FUNCTION_BLOCK ConveyorCTLMulticast (* Basic Function Block Type *)
  (* Standard: 61499-2 *)
  (* Version 0.2, 2003-12-04, JHC, Rockwell Automation, Renamed for better indexing. *)
  (* Version 0.1, 2002-11-05, JHC, Rockwell Automation, Corrected missing ST element in Algorithm REQ. *)
  (* Version 0.0, 2000-05-30, JHC, Rockwell Automation *)
  (* Compiler header: package fb.rt.cs725; *)
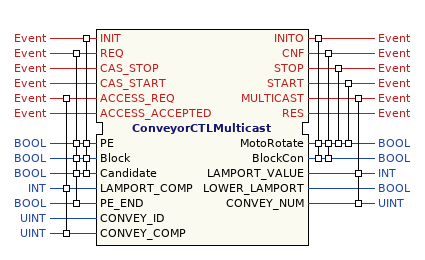
  EVENT_INPUT
    INIT WITH PE, Block, Candidate; (* Initialization Request *)
    REQ WITH PE, Block, Candidate, PE_END; (* Normal Execution Request *)
    CAS_STOP;
    CAS_START;
    ACCESS_REQ WITH LAMPORT_COMP, CONVEY_COMP;
    ACCESS_ACCEPTED;
  END_EVENT
  EVENT_OUTPUT
    INITO WITH MotoRotate, BlockCon; (* Initialization Confirm *)
    CNF WITH MotoRotate, BlockCon; (* Execution Confirmation *)
    STOP WITH MotoRotate;
    START WITH MotoRotate;
    MULTICAST WITH LAMPORT_VALUE, CONVEY_NUM;
    RES;
  END_EVENT
  VAR_INPUT
    PE : BOOL; (* Input event qualifier *)
    Block : BOOL;
    Candidate : BOOL;
    LAMPORT_COMP : INT;
    PE_END : BOOL;
    CONVEY_ID : UINT;
    CONVEY_COMP : UINT;
  END_VAR
  VAR_OUTPUT
    MotoRotate : BOOL; (* Output event qualifier *)
    BlockCon : BOOL;
    LAMPORT_VALUE : INT;
    LOWER_LAMPORT : BOOL;
    CONVEY_NUM : UINT;
  END_VAR
  VAR
    lastPE : BOOL := 1;
    lastBlock : BOOL := 0;
    LAMPORT_CLOCK : INT := 0;
  END_VAR
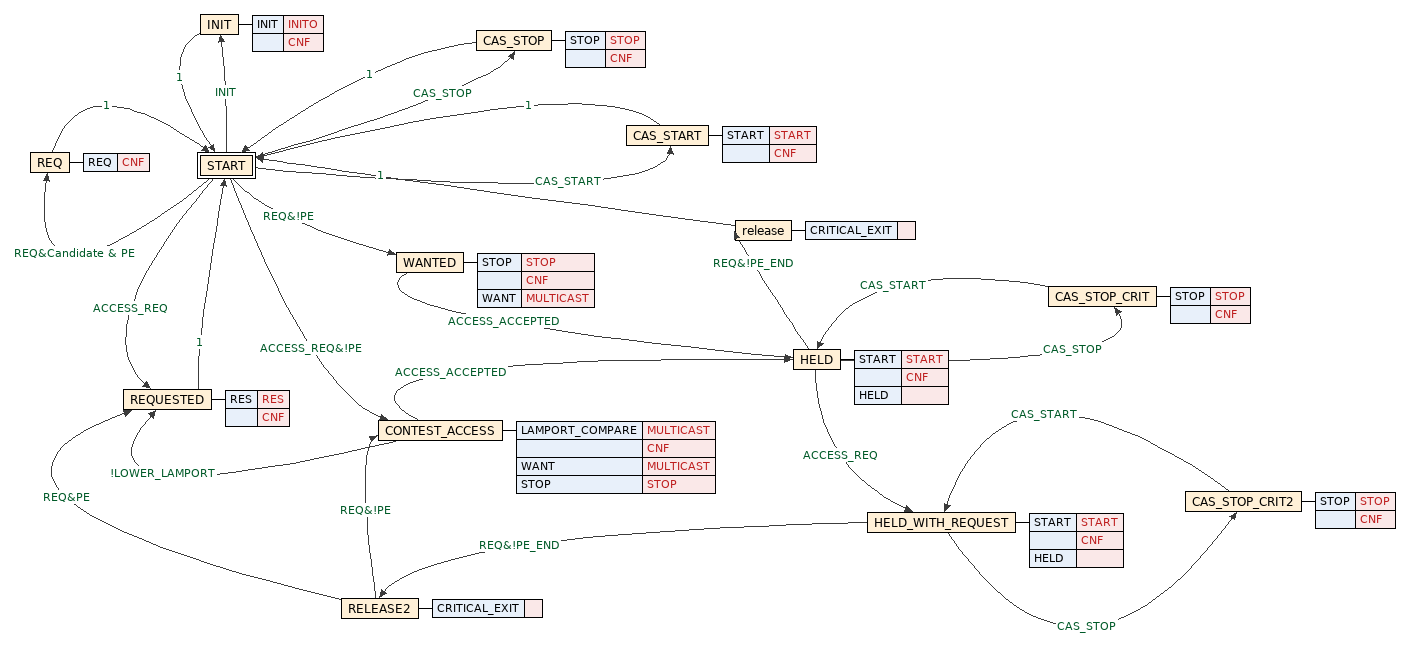
  EC_STATES
    START; (* Initial State *)
    INIT : INIT -> INITO, -> CNF; (* Initialization *)
    REQ : REQ -> CNF; (* Normal execution *)
    CAS_START : START -> START, -> CNF;
    CAS_STOP : STOP -> STOP, -> CNF;
    WANTED : STOP -> STOP, -> CNF, WANT -> MULTICAST;
    HELD : START -> START, -> CNF, HELD;
    REQUESTED : RES -> RES, -> CNF;
    CAS_STOP_CRIT : STOP -> STOP, -> CNF;
    CONTEST_ACCESS : LAMPORT_COMPARE -> MULTICAST, -> CNF, WANT -> MULTICAST, STOP -> STOP;
    release : CRITICAL_EXIT;
    HELD_WITH_REQUEST : START -> START, -> CNF, HELD;
    RELEASE2 : CRITICAL_EXIT;
    CAS_STOP_CRIT2 : STOP -> STOP, -> CNF;
  END_STATES
  EC_TRANSITIONS
    START TO INIT := INIT;
    INIT TO START := 1;
    START TO REQ := REQ&Candidate & PE;
    REQ TO START := 1;
    START TO CAS_START := CAS_START;
    CAS_START TO START := 1;
    START TO CAS_STOP := CAS_STOP;
    CAS_STOP TO START := 1;
    WANTED TO HELD := ACCESS_ACCEPTED;
    START TO WANTED := REQ&!PE;
    START TO REQUESTED := ACCESS_REQ;
    REQUESTED TO START := 1;
    CAS_STOP_CRIT TO HELD := CAS_START;
    START TO CONTEST_ACCESS := ACCESS_REQ&!PE;
    CONTEST_ACCESS TO REQUESTED := !LOWER_LAMPORT;
    CONTEST_ACCESS TO HELD := ACCESS_ACCEPTED;
    release TO START := 1;
    HELD TO release := REQ&!PE_END;
    HELD TO CAS_STOP_CRIT := CAS_STOP;
    HELD TO HELD_WITH_REQUEST := ACCESS_REQ;
    HELD_WITH_REQUEST TO CAS_STOP_CRIT2 := CAS_STOP;
    CAS_STOP_CRIT2 TO HELD_WITH_REQUEST := CAS_START;
    HELD_WITH_REQUEST TO RELEASE2 := REQ&!PE_END;
    RELEASE2 TO CONTEST_ACCESS := REQ&!PE;
    RELEASE2 TO REQUESTED := REQ&PE;
  END_TRANSITIONS
  ALGORITHM INIT IN ST: (* Initialization algorithm *)
MotoRotate := TRUE;
Block := FALSE;

System.out.println(this + " " + MotoRotate);
System.out.println(MotoRotate);
  END_ALGORITHM
  ALGORITHM REQ IN ST: (* Normally executed algorithm *)
System.out.println(CONVEY_ID +  " -> Candidate" + Candidate);
IF Candidate THEN
IF lastPE !:= PE THEN
IF NOT PE THEN
BlockCon:= TRUE;
System.out.println("BlockCon = true");
ELSE
BlockCon:=FALSE;
System.out.println("BlockCon = false");
END_IF
lastPE := PE;
END_IF
IF lastBlock !:= Block THEN
IF Block THEN
STOP.serviceEvent(this);
MotoRotate := FALSE;
System.out.println("Cas Stop");
ELSE
START.serviceEvent(this);
MotoRotate := TRUE;
System.out.println("Cas Start");
END_IF
lastBlock := Block;
END_IF
END_IF
  END_ALGORITHM
  ALGORITHM START IN Java:
MotoRotate.value=true;
System.out.println(CONVEY_ID +" Start "+MotoRotate.value);

System.out.println("Start "+MotoRotate.value);
  END_ALGORITHM
  ALGORITHM STOP IN Java:
MotoRotate.value=false;
System.out.println(CONVEY_ID +" Stop "+MotoRotate.value);

System.out.println("Stop "+MotoRotate.value);
  END_ALGORITHM
  ALGORITHM WANT IN Java:
LAMPORT_VALUE.value = LAMPORT_CLOCK.value;
System.out.println("Process "+CONVEY_ID.value + " multicasting");
System.out.println("Process "+CONVEY_ID.value + " timestamp: " + LAMPORT_CLOCK.value);
  END_ALGORITHM
  ALGORITHM LAMPORT_COMPARE IN Java:
System.out.println("Comparing Conveyor " + CONVEY_ID.value + " and " + CONVEY_COMP.value);
if (LAMPORT_COMP.value < LAMPORT_CLOCK.value) {
LOWER_LAMPORT.value = false;
}
if (LAMPORT_COMP.value == LAMPORT_CLOCK.value) {
if (CONVEY_COMP.value < CONVEY_ID.value) {
LOWER_LAMPORT.value = false;
} else {
LOWER_LAMPORT.value = true;
}
}
if (LAMPORT_COMP.value > LAMPORT_CLOCK.value) {
LOWER_LAMPORT.value = true;
}
CONVEY_NUM.value = CONVEY_ID.value;
  END_ALGORITHM
  ALGORITHM CRITICAL_EXIT IN Java:
System.out.println("Conveyor " + CONVEY_ID.value + " exited critical section");
  END_ALGORITHM
  ALGORITHM HELD IN Java:
LAMPORT_CLOCK.value++;
System.out.println("Conveyor " + CONVEY_ID.value + " accessing the critical section");
  END_ALGORITHM
  ALGORITHM RES IN Java:
System.out.println("Conveyor " + CONVEY_ID.value + " received request");
  END_ALGORITHM
END_FUNCTION_BLOCK
